FUNCTION_BLOCK DoorControl
VAR_INPUT
	PbOut1					:	BOOL;		// Pushbutton outside - door 1
	PbIn1					:	BOOL;		// Pushbutton inside - door 1
	LsDoor1Closed			:	BOOL;		// limit switch door 1 closed
	LsDoor1Opened			:	BOOL;		// limit switch door 1 opened
	
	PbOut2					:	BOOL;		// Pushbutton outside - door 2
	PbInt2					:	BOOL;		// Pushbutton inside - door 2
	LsDoor2Closed			:	BOOL;		// limit switch door 2 closed
	LsDoor2Opened			:	BOOL;		// limit switch door 2 opened
END_VAR
VAR_OUTPUT
	MotorDoor01Open			:	BOOL;		// door 1 - motor open command
	MotorDoor01Close		:	BOOL;		// door 1 - motor close command
	MotorDoor02Open			:	BOOL;		// door 2 - motor open command
	MotorDoor02Close		:	BOOL;		// door 2 - motor close command
END_VAR
VAR
	OneShot					: BOOL := TRUE;	// one shot after power recycle

	OpnSingleDoor01			: SR;			// open only door 1 request 		
	OpnDoor01Request		: SR;			// open door 1 request (door 2 following )
	OpnDoor02Request		: SR;			// open door 2 request (door 1 following)
	OpnDoor01RequestMem		: SR;			// open door 1 request memory
	OpnDoor02RequestMem		: SR;			// open door 2 request memory
	
	Wait					: SR;			// state machine: Wait	
	OpenDoor01Cmd			: SR;			// state machine: open door 1 command
	CloseDoor01Cmd			: SR;			// state machine: close door 1 command
	tonCloseDoor01Cmd		: TON;			// delay open door 1 command
	
	OpenDoor02Cmd			: SR;			// state machine: open door 2 command
	CloseDoor02Cmd			: SR;			// state machine: close door 2 command
	tonCloseDoor02Cmd		: TON;			// delay open door 2 command


	Door02Closed			: SR;			// state machine: door 1 closed
	Door01Closed			: SR;			// state machine: door 2 closed			
	
END_VAR

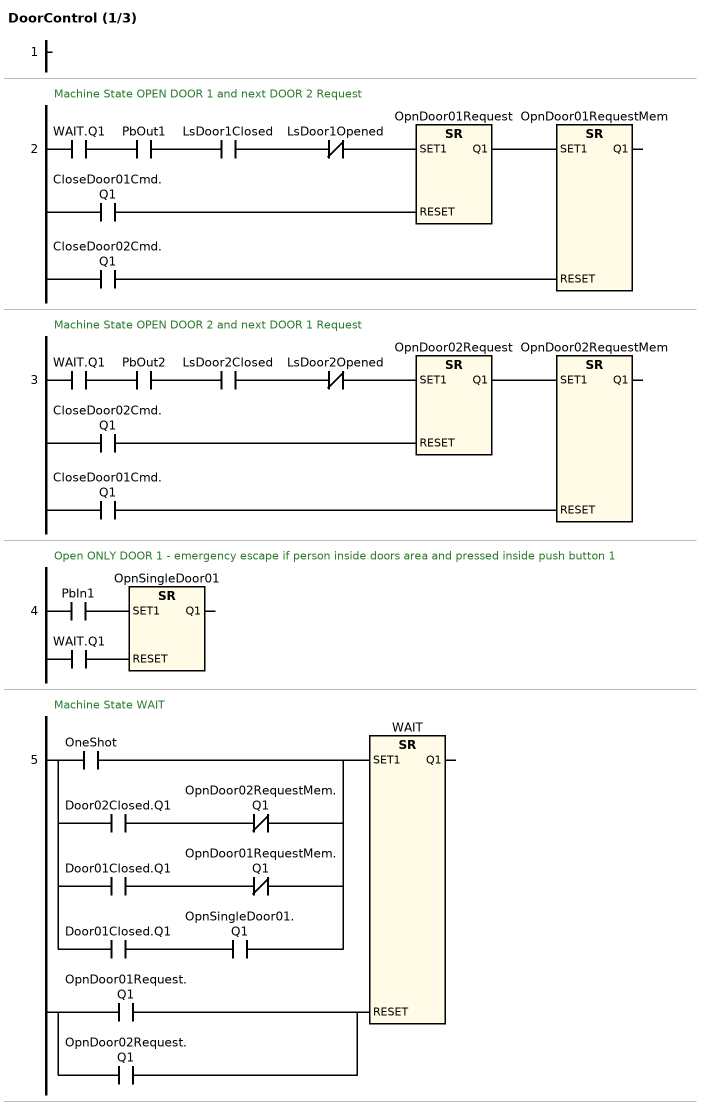
// NETWORK 1

// NETWORK 2
// Machine State OPEN DOOR 1 and next DOOR 2 Request
OpnDoor01Request(SET1 := WAIT.Q1 AND PbOut1 AND LsDoor1Closed AND NOT LsDoor1Opened, RESET := CloseDoor01Cmd.Q1); // SR
OpnDoor01RequestMem(SET1 := OpnDoor01Request.Q1, RESET := CloseDoor02Cmd.Q1); // SR

// NETWORK 3
// Machine State OPEN DOOR 2 and next DOOR 1 Request
OpnDoor02Request(SET1 := WAIT.Q1 AND PbOut2 AND LsDoor2Closed AND NOT LsDoor2Opened, RESET := CloseDoor02Cmd.Q1); // SR
OpnDoor02RequestMem(SET1 := OpnDoor02Request.Q1, RESET := CloseDoor01Cmd.Q1); // SR

// NETWORK 4
// Open ONLY DOOR 1 - emergency escape if person inside doors area and pressed inside push button 1
OpnSingleDoor01(SET1 := PbIn1, RESET := WAIT.Q1); // SR

// NETWORK 5
// Machine State WAIT
WAIT(SET1 := OneShot OR Door02Closed.Q1 AND NOT OpnDoor02RequestMem.Q1 OR Door01Closed.Q1 AND NOT OpnDoor01RequestMem.Q1 OR Door01Closed.Q1 AND OpnSingleDoor01.Q1, RESET := OpnDoor01Request.Q1 OR OpnDoor02Request.Q1); // SR

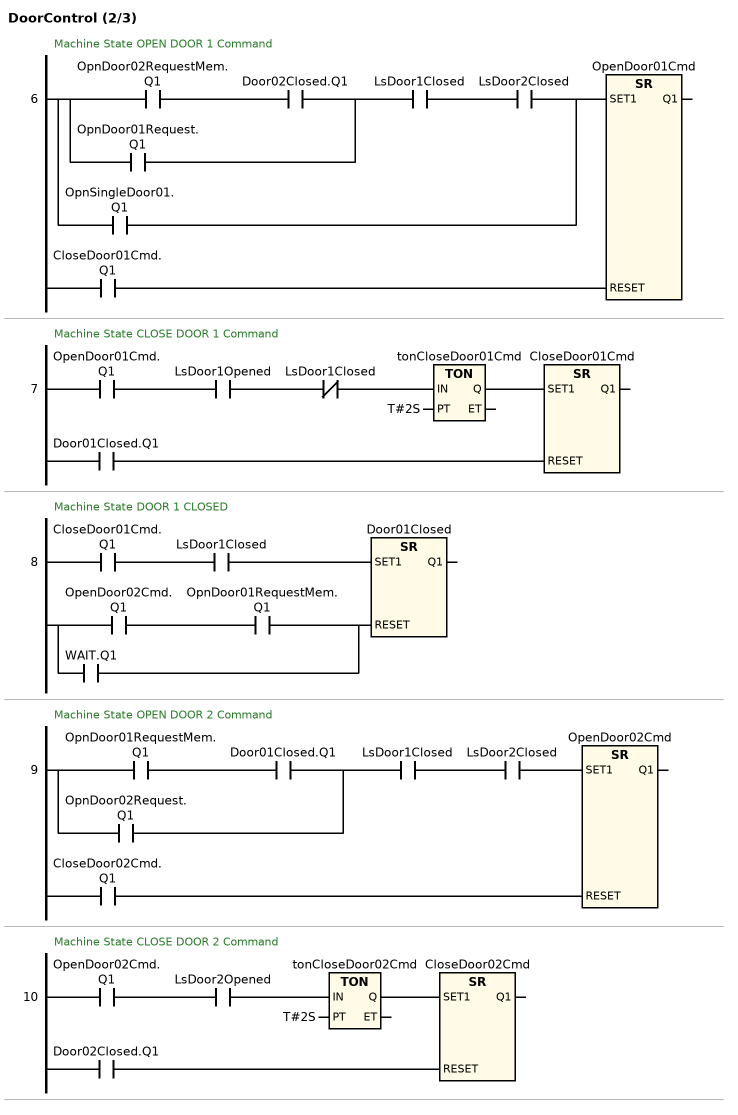
// NETWORK 6
// Machine State OPEN DOOR 1 Command
OpenDoor01Cmd(SET1 := (OpnDoor02RequestMem.Q1 AND Door02Closed.Q1 OR OpnDoor01Request.Q1) AND LsDoor1Closed AND LsDoor2Closed OR OpnSingleDoor01.Q1, RESET := CloseDoor01Cmd.Q1); // SR

// NETWORK 7
// Machine State CLOSE DOOR 1 Command
tonCloseDoor01Cmd(IN := OpenDoor01Cmd.Q1 AND LsDoor1Opened AND NOT LsDoor1Closed, PT := T#2S); // TON
CloseDoor01Cmd(SET1 := tonCloseDoor01Cmd.Q, RESET := Door01Closed.Q1); // SR

// NETWORK 8
// Machine State DOOR 1 CLOSED
Door01Closed(SET1 := CloseDoor01Cmd.Q1 AND LsDoor1Closed, RESET := OpenDoor02Cmd.Q1 AND OpnDoor01RequestMem.Q1 OR WAIT.Q1); // SR

// NETWORK 9
// Machine State OPEN DOOR 2 Command
OpenDoor02Cmd(SET1 := (OpnDoor01RequestMem.Q1 AND Door01Closed.Q1 OR OpnDoor02Request.Q1) AND LsDoor1Closed AND LsDoor2Closed, RESET := CloseDoor02Cmd.Q1); // SR

// NETWORK 10
// Machine State CLOSE DOOR 2 Command
tonCloseDoor02Cmd(IN := OpenDoor02Cmd.Q1 AND LsDoor2Opened, PT := T#2S); // TON
CloseDoor02Cmd(SET1 := tonCloseDoor02Cmd.Q, RESET := Door02Closed.Q1); // SR

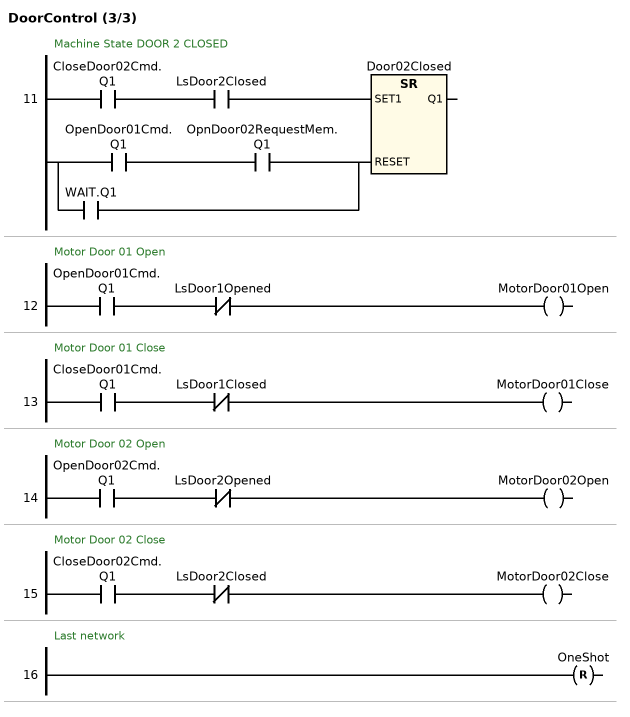
// NETWORK 11
// Machine State DOOR 2 CLOSED
Door02Closed(SET1 := CloseDoor02Cmd.Q1 AND LsDoor2Closed, RESET := OpenDoor01Cmd.Q1 AND OpnDoor02RequestMem.Q1 OR WAIT.Q1); // SR

// NETWORK 12
// Motor Door 01 Open
MotorDoor01Open := OpenDoor01Cmd.Q1 AND NOT LsDoor1Opened;

// NETWORK 13
// Motor Door 01 Close
MotorDoor01Close := CloseDoor01Cmd.Q1 AND NOT LsDoor1Closed;

// NETWORK 14
// Motor Door 02 Open
MotorDoor02Open := OpenDoor02Cmd.Q1 AND NOT LsDoor2Opened;

// NETWORK 15
// Motor Door 02 Close
MotorDoor02Close := CloseDoor02Cmd.Q1 AND NOT LsDoor2Closed;

// NETWORK 16
// Last network
OneShot R= TRUE;

END_FUNCTION_BLOCK

(* stored: Version 1.1.0.1, ProductVersion 3.1.4024.15
   POU DoorControl: Id {f8609822-686a-4d6b-934e-44f101999c27}, SpecialFunc None *)
